// TIA Portal V17 export
// export: Created 2023-02-26T22:57:58.359106Z, ExportSetting WithDefaults, DisplayName Totally Integrated Automation Portal, DisplayVersion V17, DisplayName TIA Portal Openness, DisplayVersion V17, DisplayName TIA Portal Version Control Interface, DisplayVersion V17, DisplayName TIA Portal Test Suite Advanced, DisplayVersion V17, DisplayName STEP 7 Professional, DisplayVersion V17, DisplayName SIMATIC Energy Suite, DisplayVersion V17, DisplayName STEP 7 Safety, DisplayVersion V17, DisplayName WinCC Professional, DisplayVersion V17
FUNCTION "LOG_CountPackages" : Void   // FC9, LAD
{ S7_Optimized_Access := 'TRUE' }
VERSION : 0.1
// stored: AutoNumber false, IsIECCheckEnabled false, SetENOAutomatically false, UDAEnableTagReadback false
   VAR_INPUT
      StartLine : Bool;
      ResetCountButton : Bool;
   END_VAR
   VAR_OUTPUT
      LeftCount : Int;
      ForwardCount : Int;
      RightCount : Int;
   END_VAR
   VAR_IN_OUT
      QuanitySmallPackage : Int;
      QuanityMediumPackage : Int;
      QuanityLargePackage : Int;
   END_VAR
BEGIN

REGION Network 1
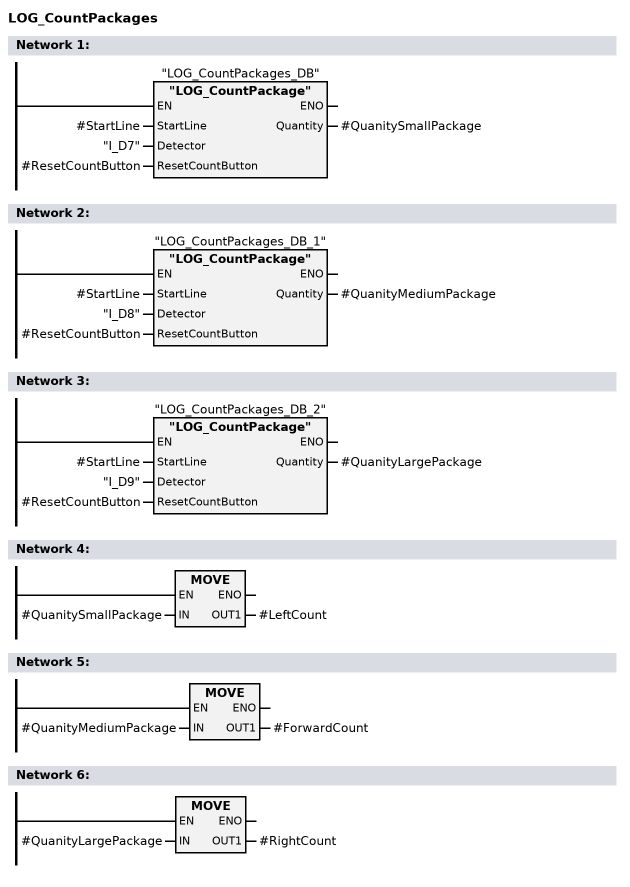
   RUNG wire#powerrail
      "LOG_CountPackages_DB"(StartLine := #StartLine, Detector := "I_D7", ResetCountButton := #ResetCountButton, Quantity => #QuanitySmallPackage)
   END_RUNG
   // the same network as SCL:
   "LOG_CountPackages_DB"(StartLine := #StartLine,   // "LOG_CountPackage"
                          Detector := "I_D7",
                          ResetCountButton := #ResetCountButton,
                          Quantity => #QuanitySmallPackage);
END_REGION

REGION Network 2
   RUNG wire#powerrail
      "LOG_CountPackages_DB_1"(StartLine := #StartLine, Detector := "I_D8", ResetCountButton := #ResetCountButton, Quantity => #QuanityMediumPackage)
   END_RUNG
   // the same network as SCL:
   "LOG_CountPackages_DB_1"(StartLine := #StartLine,   // "LOG_CountPackage"
                           Detector := "I_D8",
                           ResetCountButton := #ResetCountButton,
                           Quantity => #QuanityMediumPackage);
END_REGION

REGION Network 3
   RUNG wire#powerrail
      "LOG_CountPackages_DB_2"(StartLine := #StartLine, Detector := "I_D9", ResetCountButton := #ResetCountButton, Quantity => #QuanityLargePackage)
   END_RUNG
   // the same network as SCL:
   "LOG_CountPackages_DB_2"(StartLine := #StartLine,   // "LOG_CountPackage"
                           Detector := "I_D9",
                           ResetCountButton := #ResetCountButton,
                           Quantity => #QuanityLargePackage);
END_REGION

REGION Network 4
   RUNG wire#powerrail
      Move(in := #QuanitySmallPackage, out1 => #LeftCount)
   END_RUNG
   // the same network as SCL:
   #LeftCount := #QuanitySmallPackage;
END_REGION

REGION Network 5
   RUNG wire#powerrail
      Move(in := #QuanityMediumPackage, out1 => #ForwardCount)
   END_RUNG
   // the same network as SCL:
   #ForwardCount := #QuanityMediumPackage;
END_REGION

REGION Network 6
   RUNG wire#powerrail
      Move(in := #QuanityLargePackage, out1 => #RightCount)
   END_RUNG
   // the same network as SCL:
   #RightCount := #QuanityLargePackage;
END_REGION
END_FUNCTION
